// TIA Portal V19 export
DATA_BLOCK "INTERLOCK"   // DB117
{ S7_Optimized_Access := 'TRUE' }
// stored: MemoryReserve 100
   VAR
      ERROR : Bool;
   END_VAR
BEGIN
END_DATA_BLOCK
